Staubli VAL3: interfaceCS9.dtx

mdesc mNomSpeed
